FUNCTION_BLOCK StartFeedPosition (* Basic Function Block Type *)
  (* Standard: 61499-2 *)
  (* Version 0.0, 7/5/2026, Schneider Electric, Template *)
  PACKAGE SE.Nereda;
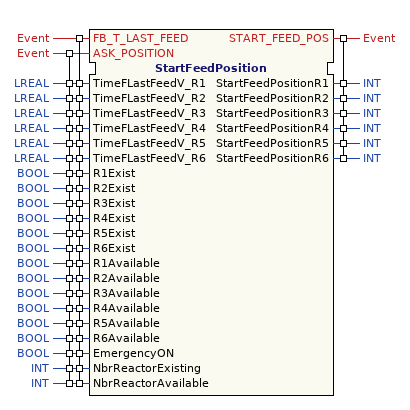
  EVENT_INPUT
    FB_T_LAST_FEED WITH TimeFLastFeedV_R1, TimeFLastFeedV_R2, TimeFLastFeedV_R3, TimeFLastFeedV_R4, TimeFLastFeedV_R5, TimeFLastFeedV_R6, R1Exist, R2Exist, R3Exist, R4Exist, R5Exist, R6Exist, R1Available, R2Available, R3Available, R4Available, R5Available, R6Available, EmergencyON, NbrReactorExisting, NbrReactorAvailable;
    ASK_POSITION WITH TimeFLastFeedV_R1, TimeFLastFeedV_R2, TimeFLastFeedV_R3, TimeFLastFeedV_R4, TimeFLastFeedV_R5, TimeFLastFeedV_R6, R1Exist, R2Exist, R3Exist, R4Exist, R5Exist, R6Exist, R1Available, R2Available, R3Available, R4Available, R5Available, R6Available, EmergencyON, NbrReactorExisting, NbrReactorAvailable;
  END_EVENT
  EVENT_OUTPUT
    START_FEED_POS WITH StartFeedPositionR1, StartFeedPositionR2, StartFeedPositionR3, StartFeedPositionR4, StartFeedPositionR5, StartFeedPositionR6;
  END_EVENT
  VAR_INPUT
    TimeFLastFeedV_R1 : LREAL;
    TimeFLastFeedV_R2 : LREAL;
    TimeFLastFeedV_R3 : LREAL;
    TimeFLastFeedV_R4 : LREAL;
    TimeFLastFeedV_R5 : LREAL;
    TimeFLastFeedV_R6 : LREAL;
    R1Exist : BOOL;
    R2Exist : BOOL;
    R3Exist : BOOL;
    R4Exist : BOOL;
    R5Exist : BOOL;
    R6Exist : BOOL;
    R1Available : BOOL;
    R2Available : BOOL;
    R3Available : BOOL;
    R4Available : BOOL;
    R5Available : BOOL;
    R6Available : BOOL;
    EmergencyON : BOOL;
    NbrReactorExisting : INT;
    NbrReactorAvailable : INT;
  END_VAR
  VAR_OUTPUT
    StartFeedPositionR1 : INT;
    StartFeedPositionR2 : INT;
    StartFeedPositionR3 : INT;
    StartFeedPositionR4 : INT;
    StartFeedPositionR5 : INT;
    StartFeedPositionR6 : INT;
  END_VAR
  VAR
    TempPosition : INT;
    FPosition : ARRAY [0..5] OF INT;
    i : INT := 0;
    ReactorOrder : ARRAY [0..5] OF INT;
  END_VAR
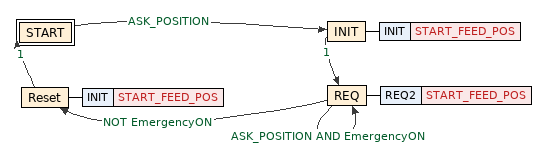
  EC_STATES
    START; (* Initial State *)
    REQ : REQ2 -> START_FEED_POS; (* Normal execution *)
    INIT : INIT -> START_FEED_POS;
    Reset : INIT -> START_FEED_POS;
  END_STATES
  EC_TRANSITIONS
    START TO INIT := ASK_POSITION;
    INIT TO REQ := 1;
    REQ TO REQ := ASK_POSITION AND EmergencyON;
    REQ TO Reset := NOT EmergencyON;
    Reset TO START := 1;
  END_TRANSITIONS
  ALGORITHM REQ IN ST: (* Normally executed algorithm *)
;
// Reset all positions at each execution
StartFeedPositionR1 := 0;
StartFeedPositionR2 := 0;
StartFeedPositionR3 := 0;
StartFeedPositionR4 := 0;
StartFeedPositionR5 := 0;
StartFeedPositionR6 := 0;


// ==================================================
// Reactor 1 position
// R1 has priority in case of equality
// ==================================================
IF R1Exist AND R1Available THEN
	StartFeedPositionR1 := 1;

	IF R2Exist AND R2Available AND (TimeFLastFeedV_R2 > TimeFLastFeedV_R1) THEN
		StartFeedPositionR1 := StartFeedPositionR1 + 1;
	END_IF;

	IF R3Exist AND R3Available AND (TimeFLastFeedV_R3 > TimeFLastFeedV_R1) THEN
		StartFeedPositionR1 := StartFeedPositionR1 + 1;
	END_IF;

	IF R4Exist AND R4Available AND (TimeFLastFeedV_R4 > TimeFLastFeedV_R1) THEN
		StartFeedPositionR1 := StartFeedPositionR1 + 1;
	END_IF;

	IF R5Exist AND R5Available AND (TimeFLastFeedV_R5 > TimeFLastFeedV_R1) THEN
		StartFeedPositionR1 := StartFeedPositionR1 + 1;
	END_IF;

	IF R6Exist AND R6Available AND (TimeFLastFeedV_R6 > TimeFLastFeedV_R1) THEN
		StartFeedPositionR1 := StartFeedPositionR1 + 1;
	END_IF;
END_IF;


// ==================================================
// Reactor 2 position
// R1 has priority over R2 in case of equality
// ==================================================
IF R2Exist AND R2Available THEN
	StartFeedPositionR2 := 1;

	IF R1Exist AND R1Available AND (TimeFLastFeedV_R1 >= TimeFLastFeedV_R2) THEN
		StartFeedPositionR2 := StartFeedPositionR2 + 1;
	END_IF;

	IF R3Exist AND R3Available AND (TimeFLastFeedV_R3 > TimeFLastFeedV_R2) THEN
		StartFeedPositionR2 := StartFeedPositionR2 + 1;
	END_IF;

	IF R4Exist AND R4Available AND (TimeFLastFeedV_R4 > TimeFLastFeedV_R2) THEN
		StartFeedPositionR2 := StartFeedPositionR2 + 1;
	END_IF;

	IF R5Exist AND R5Available AND (TimeFLastFeedV_R5 > TimeFLastFeedV_R2) THEN
		StartFeedPositionR2 := StartFeedPositionR2 + 1;
	END_IF;

	IF R6Exist AND R6Available AND (TimeFLastFeedV_R6 > TimeFLastFeedV_R2) THEN
		StartFeedPositionR2 := StartFeedPositionR2 + 1;
	END_IF;
END_IF;


// ==================================================
// Reactor 3 position
// R1 and R2 have priority over R3 in case of equality
// ==================================================
IF R3Exist AND R3Available THEN
	StartFeedPositionR3 := 1;

	IF R1Exist AND R1Available AND (TimeFLastFeedV_R1 >= TimeFLastFeedV_R3) THEN
		StartFeedPositionR3 := StartFeedPositionR3 + 1;
	END_IF;

	IF R2Exist AND R2Available AND (TimeFLastFeedV_R2 >= TimeFLastFeedV_R3) THEN
		StartFeedPositionR3 := StartFeedPositionR3 + 1;
	END_IF;

	IF R4Exist AND R4Available AND (TimeFLastFeedV_R4 > TimeFLastFeedV_R3) THEN
		StartFeedPositionR3 := StartFeedPositionR3 + 1;
	END_IF;

	IF R5Exist AND R5Available AND (TimeFLastFeedV_R5 > TimeFLastFeedV_R3) THEN
		StartFeedPositionR3 := StartFeedPositionR3 + 1;
	END_IF;

	IF R6Exist AND R6Available AND (TimeFLastFeedV_R6 > TimeFLastFeedV_R3) THEN
		StartFeedPositionR3 := StartFeedPositionR3 + 1;
	END_IF;
END_IF;


// ==================================================
// Reactor 4 position
// R1, R2 and R3 have priority over R4 in case of equality
// ==================================================
IF R4Exist AND R4Available THEN
	StartFeedPositionR4 := 1;

	IF R1Exist AND R1Available AND (TimeFLastFeedV_R1 >= TimeFLastFeedV_R4) THEN
		StartFeedPositionR4 := StartFeedPositionR4 + 1;
	END_IF;

	IF R2Exist AND R2Available AND (TimeFLastFeedV_R2 >= TimeFLastFeedV_R4) THEN
		StartFeedPositionR4 := StartFeedPositionR4 + 1;
	END_IF;

	IF R3Exist AND R3Available AND (TimeFLastFeedV_R3 >= TimeFLastFeedV_R4) THEN
		StartFeedPositionR4 := StartFeedPositionR4 + 1;
	END_IF;

	IF R5Exist AND R5Available AND (TimeFLastFeedV_R5 > TimeFLastFeedV_R4) THEN
		StartFeedPositionR4 := StartFeedPositionR4 + 1;
	END_IF;

	IF R6Exist AND R6Available AND (TimeFLastFeedV_R6 > TimeFLastFeedV_R4) THEN
		StartFeedPositionR4 := StartFeedPositionR4 + 1;
	END_IF;
END_IF;


// ==================================================
// Reactor 5 position
// R1, R2, R3 and R4 have priority over R5 in case of equality
// ==================================================
IF R5Exist AND R5Available THEN
	StartFeedPositionR5 := 1;

	IF R1Exist AND R1Available AND (TimeFLastFeedV_R1 >= TimeFLastFeedV_R5) THEN
		StartFeedPositionR5 := StartFeedPositionR5 + 1;
	END_IF;

	IF R2Exist AND R2Available AND (TimeFLastFeedV_R2 >= TimeFLastFeedV_R5) THEN
		StartFeedPositionR5 := StartFeedPositionR5 + 1;
	END_IF;

	IF R3Exist AND R3Available AND (TimeFLastFeedV_R3 >= TimeFLastFeedV_R5) THEN
		StartFeedPositionR5 := StartFeedPositionR5 + 1;
	END_IF;

	IF R4Exist AND R4Available AND (TimeFLastFeedV_R4 >= TimeFLastFeedV_R5) THEN
		StartFeedPositionR5 := StartFeedPositionR5 + 1;
	END_IF;

	IF R6Exist AND R6Available AND (TimeFLastFeedV_R6 > TimeFLastFeedV_R5) THEN
		StartFeedPositionR5 := StartFeedPositionR5 + 1;
	END_IF;
END_IF;


// ==================================================
// Reactor 6 position
// R1, R2, R3, R4 and R5 have priority over R6 in case of equality
// ==================================================
IF R6Exist AND R6Available THEN
	StartFeedPositionR6 := 1;

	IF R1Exist AND R1Available AND (TimeFLastFeedV_R1 >= TimeFLastFeedV_R6) THEN
		StartFeedPositionR6 := StartFeedPositionR6 + 1;
	END_IF;

	IF R2Exist AND R2Available AND (TimeFLastFeedV_R2 >= TimeFLastFeedV_R6) THEN
		StartFeedPositionR6 := StartFeedPositionR6 + 1;
	END_IF;

	IF R3Exist AND R3Available AND (TimeFLastFeedV_R3 >= TimeFLastFeedV_R6) THEN
		StartFeedPositionR6 := StartFeedPositionR6 + 1;
	END_IF;

	IF R4Exist AND R4Available AND (TimeFLastFeedV_R4 >= TimeFLastFeedV_R6) THEN
		StartFeedPositionR6 := StartFeedPositionR6 + 1;
	END_IF;

	IF R5Exist AND R5Available AND (TimeFLastFeedV_R5 >= TimeFLastFeedV_R6) THEN
		StartFeedPositionR6 := StartFeedPositionR6 + 1;
	END_IF;
END_IF;

FPosition[0] := StartFeedPositionR1;
FPosition[1] := StartFeedPositionR2;
FPosition[2] := StartFeedPositionR3;
FPosition[3] := StartFeedPositionR4;
FPosition[4] := StartFeedPositionR5;
FPosition[5] := StartFeedPositionR6;

ASK_POSITION := FALSE;
  END_ALGORITHM
  ALGORITHM INIT IN ST:
;
// Reset all positions at each execution
StartFeedPositionR1 := 0;
StartFeedPositionR2 := 0;
StartFeedPositionR3 := 0;
StartFeedPositionR4 := 0;
StartFeedPositionR5 := 0;
StartFeedPositionR6 := 0;
  END_ALGORITHM
  ALGORITHM RxUnAv IN ST:
;
IF NOT R1Available AND R1Exist THEN
	FPosition[0] := NbrReactorExisting;
END_IF;

IF NOT R2Available AND R2Exist THEN
	FPosition[1] := NbrReactorExisting;
END_IF;

IF NOT R3Available AND R3Exist THEN
	FPosition[2] := NbrReactorExisting;
END_IF;

IF NOT R4Available AND R4Exist THEN
	FPosition[3] := NbrReactorExisting;
END_IF;

IF NOT R5Available AND R5Exist THEN
	FPosition[4] := NbrReactorExisting;
END_IF;

IF NOT R6Available AND R6Exist THEN
	FPosition[5] := NbrReactorExisting;
END_IF;

TempPosition := FPosition[0];

FOR i := 0 TO NbrReactorExisting - (2 + NbrReactorExisting - NbrReactorAvailable) DO
    FPosition[i] := FPosition[i + 1];
END_FOR;

FPosition[NbrReactorExisting - (1 + NbrReactorExisting - NbrReactorAvailable)] := TempPosition;

StartFeedPositionR1 := FPosition[0];
StartFeedPositionR2 := FPosition[1];
StartFeedPositionR3 := FPosition[2];
StartFeedPositionR4 := FPosition[3];
StartFeedPositionR5 := FPosition[4];
StartFeedPositionR6 := FPosition[5];

ASK_POSITION := FALSE;
  END_ALGORITHM
  ALGORITHM InitRxUnAv IN ST:
;
// Reset all positions at each execution
FPosition[0] := 0;
FPosition[1] := 0;
FPosition[2] := 0;
FPosition[3] := 0;
FPosition[4] := 0;
FPosition[5] := 0;

// ==================================================
// Reactor 1 position
// R1 has priority in case of equality
// ==================================================
IF R1Exist AND R1Available THEN
    FPosition[0] := 1;

    IF R2Exist AND R2Available AND (TimeFLastFeedV_R2 > TimeFLastFeedV_R1) THEN
        FPosition[0] := FPosition[0] + 1;
    END_IF;

    IF R3Exist AND R3Available AND (TimeFLastFeedV_R3 > TimeFLastFeedV_R1) THEN
        FPosition[0] := FPosition[0] + 1;
    END_IF;

    IF R4Exist AND R4Available AND (TimeFLastFeedV_R4 > TimeFLastFeedV_R1) THEN
        FPosition[0] := FPosition[0] + 1;
    END_IF;

    IF R5Exist AND R5Available AND (TimeFLastFeedV_R5 > TimeFLastFeedV_R1) THEN
        FPosition[0] := FPosition[0] + 1;
    END_IF;

    IF R6Exist AND R6Available AND (TimeFLastFeedV_R6 > TimeFLastFeedV_R1) THEN
        FPosition[0] := FPosition[0] + 1;
    END_IF;

END_IF;

// ==================================================
// Reactor 2 position
// R1 has priority over R2 in case of equality
// ==================================================
IF R2Exist AND R2Available THEN
    FPosition[1] := 1;

    IF R1Exist AND R1Available AND (TimeFLastFeedV_R1 >= TimeFLastFeedV_R2) THEN
        FPosition[1] := FPosition[1] + 1;
    END_IF;

    IF R3Exist AND R3Available AND (TimeFLastFeedV_R3 > TimeFLastFeedV_R2) THEN
        FPosition[1] := FPosition[1] + 1;
    END_IF;

    IF R4Exist AND R4Available AND (TimeFLastFeedV_R4 > TimeFLastFeedV_R2) THEN
        FPosition[1] := FPosition[1] + 1;
    END_IF;

    IF R5Exist AND R5Available AND (TimeFLastFeedV_R5 > TimeFLastFeedV_R2) THEN
        FPosition[1] := FPosition[1] + 1;
    END_IF;

    IF R6Exist AND R6Available AND (TimeFLastFeedV_R6 > TimeFLastFeedV_R2) THEN
        FPosition[1] := FPosition[1] + 1;
    END_IF;

END_IF;

// ==================================================
// Reactor 3 position
// ==================================================
IF R3Exist AND R3Available THEN
    FPosition[2] := 1;

    IF R1Exist AND R1Available AND (TimeFLastFeedV_R1 >= TimeFLastFeedV_R3) THEN
        FPosition[2] := FPosition[2] + 1;
    END_IF;

    IF R2Exist AND R2Available AND (TimeFLastFeedV_R2 >= TimeFLastFeedV_R3) THEN
        FPosition[2] := FPosition[2] + 1;
    END_IF;

    IF R4Exist AND R4Available AND (TimeFLastFeedV_R4 > TimeFLastFeedV_R3) THEN
        FPosition[2] := FPosition[2] + 1;
    END_IF;

    IF R5Exist AND R5Available AND (TimeFLastFeedV_R5 > TimeFLastFeedV_R3) THEN
        FPosition[2] := FPosition[2] + 1;
    END_IF;

    IF R6Exist AND R6Available AND (TimeFLastFeedV_R6 > TimeFLastFeedV_R3) THEN
        FPosition[2] := FPosition[2] + 1;
    END_IF;

END_IF;

// ==================================================
// Reactor 4 position
// ==================================================
IF R4Exist AND R4Available THEN
    FPosition[3] := 1;

    IF R1Exist AND R1Available AND (TimeFLastFeedV_R1 >= TimeFLastFeedV_R4) THEN
        FPosition[3] := FPosition[3] + 1;
    END_IF;

    IF R2Exist AND R2Available AND (TimeFLastFeedV_R2 >= TimeFLastFeedV_R4) THEN
        FPosition[3] := FPosition[3] + 1;
    END_IF;

    IF R3Exist AND R3Available AND (TimeFLastFeedV_R3 >= TimeFLastFeedV_R4) THEN
        FPosition[3] := FPosition[3] + 1;
    END_IF;

    IF R5Exist AND R5Available AND (TimeFLastFeedV_R5 > TimeFLastFeedV_R4) THEN
        FPosition[3] := FPosition[3] + 1;
    END_IF;

    IF R6Exist AND R6Available AND (TimeFLastFeedV_R6 > TimeFLastFeedV_R4) THEN
        FPosition[3] := FPosition[3] + 1;
    END_IF;

END_IF;

// ==================================================
// Reactor 5 position
// ==================================================
IF R5Exist AND R5Available THEN
    FPosition[4] := 1;

    IF R1Exist AND R1Available AND (TimeFLastFeedV_R1 >= TimeFLastFeedV_R5) THEN
        FPosition[4] := FPosition[4] + 1;
    END_IF;

    IF R2Exist AND R2Available AND (TimeFLastFeedV_R2 >= TimeFLastFeedV_R5) THEN
        FPosition[4] := FPosition[4] + 1;
    END_IF;

    IF R3Exist AND R3Available AND (TimeFLastFeedV_R3 >= TimeFLastFeedV_R5) THEN
        FPosition[4] := FPosition[4] + 1;
    END_IF;

    IF R4Exist AND R4Available AND (TimeFLastFeedV_R4 >= TimeFLastFeedV_R5) THEN
        FPosition[4] := FPosition[4] + 1;
    END_IF;

    IF R6Exist AND R6Available AND (TimeFLastFeedV_R6 > TimeFLastFeedV_R5) THEN
        FPosition[4] := FPosition[4] + 1;
    END_IF;

END_IF;

// ==================================================
// Reactor 6 position
// ==================================================
IF R6Exist AND R6Available THEN
    FPosition[5] := 1;

    IF R1Exist AND R1Available AND (TimeFLastFeedV_R1 >= TimeFLastFeedV_R6) THEN
        FPosition[5] := FPosition[5] + 1;
    END_IF;

    IF R2Exist AND R2Available AND (TimeFLastFeedV_R2 >= TimeFLastFeedV_R6) THEN
        FPosition[5] := FPosition[5] + 1;
    END_IF;

    IF R3Exist AND R3Available AND (TimeFLastFeedV_R3 >= TimeFLastFeedV_R6) THEN
        FPosition[5] := FPosition[5] + 1;
    END_IF;

    IF R4Exist AND R4Available AND (TimeFLastFeedV_R4 >= TimeFLastFeedV_R6) THEN
        FPosition[5] := FPosition[5] + 1;
    END_IF;

    IF R5Exist AND R5Available AND (TimeFLastFeedV_R5 >= TimeFLastFeedV_R6) THEN
        FPosition[5] := FPosition[5] + 1;
    END_IF;

END_IF;
  END_ALGORITHM
  ALGORITHM REQ2 IN ST:
;
// Reset all positions at each execution
StartFeedPositionR1 := 0;
StartFeedPositionR2 := 0;
StartFeedPositionR3 := 0;
StartFeedPositionR4 := 0;
StartFeedPositionR5 := 0;
StartFeedPositionR6 := 0;


// ==================================================
// Reactor 1 position
// ==================================================
IF R1Exist AND R1Available THEN

    StartFeedPositionR1 := 1;

    IF R2Exist AND R2Available AND (TimeFLastFeedV_R2 > TimeFLastFeedV_R1) THEN
        StartFeedPositionR1 := StartFeedPositionR1 + 1;
    END_IF;

    IF R3Exist AND R3Available AND (TimeFLastFeedV_R3 > TimeFLastFeedV_R1) THEN
        StartFeedPositionR1 := StartFeedPositionR1 + 1;
    END_IF;

    IF R4Exist AND R4Available AND (TimeFLastFeedV_R4 > TimeFLastFeedV_R1) THEN
        StartFeedPositionR1 := StartFeedPositionR1 + 1;
    END_IF;

    IF R5Exist AND R5Available AND (TimeFLastFeedV_R5 > TimeFLastFeedV_R1) THEN
        StartFeedPositionR1 := StartFeedPositionR1 + 1;
    END_IF;

    IF R6Exist AND R6Available AND (TimeFLastFeedV_R6 > TimeFLastFeedV_R1) THEN
        StartFeedPositionR1 := StartFeedPositionR1 + 1;
    END_IF;

ELSIF R1Exist AND NOT R1Available THEN

    StartFeedPositionR1 := NbrReactorExisting;

END_IF;


// ==================================================
// Reactor 2 position
// ==================================================
IF R2Exist AND R2Available THEN

    StartFeedPositionR2 := 1;

    IF R1Exist AND R1Available AND (TimeFLastFeedV_R1 >= TimeFLastFeedV_R2) THEN
        StartFeedPositionR2 := StartFeedPositionR2 + 1;
    END_IF;

    IF R3Exist AND R3Available AND (TimeFLastFeedV_R3 > TimeFLastFeedV_R2) THEN
        StartFeedPositionR2 := StartFeedPositionR2 + 1;
    END_IF;

    IF R4Exist AND R4Available AND (TimeFLastFeedV_R4 > TimeFLastFeedV_R2) THEN
        StartFeedPositionR2 := StartFeedPositionR2 + 1;
    END_IF;

    IF R5Exist AND R5Available AND (TimeFLastFeedV_R5 > TimeFLastFeedV_R2) THEN
        StartFeedPositionR2 := StartFeedPositionR2 + 1;
    END_IF;

    IF R6Exist AND R6Available AND (TimeFLastFeedV_R6 > TimeFLastFeedV_R2) THEN
        StartFeedPositionR2 := StartFeedPositionR2 + 1;
    END_IF;

ELSIF R2Exist AND NOT R2Available THEN

    StartFeedPositionR2 := NbrReactorExisting;

END_IF;


// ==================================================
// Reactor 3 position
// ==================================================
IF R3Exist AND R3Available THEN

    StartFeedPositionR3 := 1;

    IF R1Exist AND R1Available AND (TimeFLastFeedV_R1 >= TimeFLastFeedV_R3) THEN
        StartFeedPositionR3 := StartFeedPositionR3 + 1;
    END_IF;

    IF R2Exist AND R2Available AND (TimeFLastFeedV_R2 >= TimeFLastFeedV_R3) THEN
        StartFeedPositionR3 := StartFeedPositionR3 + 1;
    END_IF;

    IF R4Exist AND R4Available AND (TimeFLastFeedV_R4 > TimeFLastFeedV_R3) THEN
        StartFeedPositionR3 := StartFeedPositionR3 + 1;
    END_IF;

    IF R5Exist AND R5Available AND (TimeFLastFeedV_R5 > TimeFLastFeedV_R3) THEN
        StartFeedPositionR3 := StartFeedPositionR3 + 1;
    END_IF;

    IF R6Exist AND R6Available AND (TimeFLastFeedV_R6 > TimeFLastFeedV_R3) THEN
        StartFeedPositionR3 := StartFeedPositionR3 + 1;
    END_IF;

ELSIF R3Exist AND NOT R3Available THEN

    StartFeedPositionR3 := NbrReactorExisting;

END_IF;


// ==================================================
// Reactor 4 position
// ==================================================
IF R4Exist AND R4Available THEN

    StartFeedPositionR4 := 1;

    IF R1Exist AND R1Available AND (TimeFLastFeedV_R1 >= TimeFLastFeedV_R4) THEN
        StartFeedPositionR4 := StartFeedPositionR4 + 1;
    END_IF;

    IF R2Exist AND R2Available AND (TimeFLastFeedV_R2 >= TimeFLastFeedV_R4) THEN
        StartFeedPositionR4 := StartFeedPositionR4 + 1;
    END_IF;

    IF R3Exist AND R3Available AND (TimeFLastFeedV_R3 >= TimeFLastFeedV_R4) THEN
        StartFeedPositionR4 := StartFeedPositionR4 + 1;
    END_IF;

    IF R5Exist AND R5Available AND (TimeFLastFeedV_R5 > TimeFLastFeedV_R4) THEN
        StartFeedPositionR4 := StartFeedPositionR4 + 1;
    END_IF;

    IF R6Exist AND R6Available AND (TimeFLastFeedV_R6 > TimeFLastFeedV_R4) THEN
        StartFeedPositionR4 := StartFeedPositionR4 + 1;
    END_IF;

ELSIF R4Exist AND NOT R4Available THEN

    StartFeedPositionR4 := NbrReactorExisting;

END_IF;


// ==================================================
// Reactor 5 position
// ==================================================
IF R5Exist AND R5Available THEN

    StartFeedPositionR5 := 1;

    IF R1Exist AND R1Available AND (TimeFLastFeedV_R1 >= TimeFLastFeedV_R5) THEN
        StartFeedPositionR5 := StartFeedPositionR5 + 1;
    END_IF;

    IF R2Exist AND R2Available AND (TimeFLastFeedV_R2 >= TimeFLastFeedV_R5) THEN
        StartFeedPositionR5 := StartFeedPositionR5 + 1;
    END_IF;

    IF R3Exist AND R3Available AND (TimeFLastFeedV_R3 >= TimeFLastFeedV_R5) THEN
        StartFeedPositionR5 := StartFeedPositionR5 + 1;
    END_IF;

    IF R4Exist AND R4Available AND (TimeFLastFeedV_R4 >= TimeFLastFeedV_R5) THEN
        StartFeedPositionR5 := StartFeedPositionR5 + 1;
    END_IF;

    IF R6Exist AND R6Available AND (TimeFLastFeedV_R6 > TimeFLastFeedV_R5) THEN
        StartFeedPositionR5 := StartFeedPositionR5 + 1;
    END_IF;

ELSIF R5Exist AND NOT R5Available THEN

    StartFeedPositionR5 := NbrReactorExisting;

END_IF;


// ==================================================
// Reactor 6 position
// ==================================================
IF R6Exist AND R6Available THEN

    StartFeedPositionR6 := 1;

    IF R1Exist AND R1Available AND (TimeFLastFeedV_R1 >= TimeFLastFeedV_R6) THEN
        StartFeedPositionR6 := StartFeedPositionR6 + 1;
    END_IF;

    IF R2Exist AND R2Available AND (TimeFLastFeedV_R2 >= TimeFLastFeedV_R6) THEN
        StartFeedPositionR6 := StartFeedPositionR6 + 1;
    END_IF;

    IF R3Exist AND R3Available AND (TimeFLastFeedV_R3 >= TimeFLastFeedV_R6) THEN
        StartFeedPositionR6 := StartFeedPositionR6 + 1;
    END_IF;

    IF R4Exist AND R4Available AND (TimeFLastFeedV_R4 >= TimeFLastFeedV_R6) THEN
        StartFeedPositionR6 := StartFeedPositionR6 + 1;
    END_IF;

    IF R5Exist AND R5Available AND (TimeFLastFeedV_R5 >= TimeFLastFeedV_R6) THEN
        StartFeedPositionR6 := StartFeedPositionR6 + 1;
    END_IF;

ELSIF R6Exist AND NOT R6Available THEN

    StartFeedPositionR6 := NbrReactorExisting;

END_IF;
  END_ALGORITHM
END_FUNCTION_BLOCK
